// TIA Portal V17 export
// export: Created 2024-09-03T21:54:49.5214082Z, ExportSetting WithDefaults, DisplayName Totally Integrated Automation Portal, DisplayVersion V17 Update 7, DisplayName TIA Portal Openness, DisplayVersion V17 Update 7, DisplayName TIA Portal Version Control Interface, DisplayVersion V17, DisplayName SINAMICS Startdrive Advanced, DisplayVersion V17 SP2, DisplayName SINAMICS Startdrive G110M, G120, G120C, G120D, G120P, G115D, DisplayVersion V17 SP2, DisplayName SINAMICS Startdrive G130, G150, S120, S150, SINAMICS MV, S210, DisplayVersion V17 SP2, DisplayName STEP 7 Professional, DisplayVersion V17 Update 7, DisplayName STEP 7 Safety, DisplayVersion V17 Update 6, DisplayName WinCC Advanced / Unified PC, DisplayVersion V17 Update 7
DATA_BLOCK "FittingHistoryRightCupforming_DB"   // DB43
VERSION : 0.1
// stored: AutoNumber true, DBAccessibleFromOPCUA true, DBAccessibleFromWebserver true, InstanceOfName FittingHistory, InstanceOfType FB
"FittingHistory"
   // VAR_INPUT
   //    iNewCycle : Bool;
   //    iData : "UDT_Results_Cupforming";
   // END_VAR
   // VAR RETAIN
   //    history : Array[0..99] of "UDT_Results_Cupforming";
   // END_VAR
   // VAR
   //    pageData { S7_SetPoint := 'True'} : Array[0..9] of "UDT_Results_Cupforming";
   // END_VAR
   // VAR RETAIN
   //    pageNumber { S7_SetPoint := 'True'} : USInt := 0;
   // END_VAR
   // VAR
   //    resetHistory : Bool;
   //    R_TRIG_Instance { S7_SetPoint := 'True'} : R_TRIG;
   // END_VAR
BEGIN
   history[0].MaxForce := 8.163286;
   history[1].MaxForce := 8.130146;
   history[2..3].MaxForce := 8.158552;
   history[4..5].MaxForce := 8.177489;
   history[6].MaxForce := 8.149084;
   history[7].MaxForce := 8.158552;
   history[8].MaxForce := 54.72517;
   history[9].MaxForce := 54.91927;
   history[10].MaxForce := 52.27753;
   history[11..99].MaxForce := 0.0;
   history[0].MinimalWay := 9.87697;
   history[1].MinimalWay := 9.87257;
   history[2].MinimalWay := 9.886649;
   history[3].MinimalWay := 9.885769;
   history[4].MinimalWay := 9.896328;
   history[5].MinimalWay := 9.890168;
   history[6].MinimalWay := 9.88137;
   history[7].MinimalWay := 9.887528;
   history[8].MinimalWay := 9.091208;
   history[9].MinimalWay := 8.947783;
   history[10].MinimalWay := 8.997938;
   history[11..99].MinimalWay := 0.0;
   history[0].MaxZposition := 56.52127;
   history[1].MaxZposition := 56.64497;
   history[2].MaxZposition := 56.6059;
   history[3].MaxZposition := 56.54731;
   history[4].MaxZposition := 56.57769;
   history[5].MaxZposition := 56.63412;
   history[6].MaxZposition := 56.4974;
   history[7].MaxZposition := 56.69054;
   history[8].MaxZposition := 58.5612;
   history[9].MaxZposition := 58.33334;
   history[10].MaxZposition := 58.6849;
   history[11..99].MaxZposition := 0.0;
   history[0..10].OK := TRUE;
   history[11..99].OK := FALSE;
   history[0..99].NOK := FALSE;
   history[0..10].parameters.DigiforceProgram := 1;
   history[11..99].parameters.DigiforceProgram := 0;
   history[0..10].parameters.FinalSpeed := 20.0;
   history[11..99].parameters.FinalSpeed := 0.0;
   history[0..10].parameters.ApproachSpeed := 100.0;
   history[11..99].parameters.ApproachSpeed := 0.0;
   history[0..7].parameters.FinalForce := 80.0;
   history[8..10].parameters.FinalForce := 90.0;
   history[11..99].parameters.FinalForce := 0.0;
   history[0..10].parameters.ApproachForce := 20.0;
   history[11..99].parameters.ApproachForce := 0.0;
   history[0..7].parameters.EndWayImmediate := 9.9;
   history[8..10].parameters.EndWayImmediate := 9.0;
   history[11..99].parameters.EndWayImmediate := 0.0;
   history[0..7].parameters.EndWayWithTimeout := 9.9;
   history[8..9].parameters.EndWayWithTimeout := 9.1;
   history[10].parameters.EndWayWithTimeout := 9.0;
   history[11..99].parameters.EndWayWithTimeout := 0.0;
   history[0..7].parameters.SwitchingWay := 50.0;
   history[8..10].parameters.SwitchingWay := 53.0;
   history[11..99].parameters.SwitchingWay := 0.0;
   history[0..10].parameters.EndWayTimeout := T#300MS;
   history[11..99].parameters.EndWayTimeout := T#0MS;
END_DATA_BLOCK
